{attribute addProperty BoxType "EJ3202-0000-0019"}
{attribute addProperty Id "StatusAT %I*Status_C6F82E6F658.1251ValueAT %I*INT16217"}
{attribute addProperty CRC "3038476796"}
{attribute addProperty SizeInBites "81"}
{attribute addProperty SizeInBytes "10.125"}
TYPE RTD_Inputs_Channel_B51B79FC :
STRUCT
	{attribute addProperty Name "Status"}
	Status AT %I* : Status_C6F82E6F;
	{attribute addProperty Name "Value"}
	Value AT %I* : INT;
END_STRUCT
END_TYPE

(* stored: Version 1.2.0.0, ProductVersion 3.1.4024.9
   DUT RTD_Inputs_Channel_B51B79FC: Id {1496a16d-464b-451c-a730-86aafc126dfd} *)
